// TIA Portal V17 export
// export: Created 2026-05-13T16:54:41.5069404Z, ExportSetting WithDefaults, DisplayName Totally Integrated Automation Portal, DisplayVersion V17 Update 4, DisplayName TIA Portal Openness, DisplayVersion V17 Update 4, DisplayName TIA Portal Version Control Interface, DisplayVersion V17, DisplayName SINAMICS Startdrive Advanced, DisplayVersion V17, DisplayName SINAMICS Startdrive G130, G150, S120, S150, SINAMICS MV, S210, DisplayVersion V17, DisplayName SINAMICS Startdrive G110M, G120, G120C, G120D, G120P, G115D, DisplayVersion V17, DisplayName STEP 7 Professional, DisplayVersion V17 Update 4, DisplayName STEP 7 Safety, DisplayVersion V17, DisplayName WinCC Professional, DisplayVersion V17 Update 4
TagTable "SV"
  SV_BD布袋压差高报 : Real  (PLC tag SV.BD布袋压差高报, HMI_连接_1, 1 s)
  SV_BD布袋压差高高报 : Real  (PLC tag SV.BD布袋压差高高报, HMI_连接_1, 1 s)
  SV_GX高效压差高报 : Real  (PLC tag SV.GX高效压差高报, HMI_连接_1, 1 s)
  SV_GX高效压差高高报 : Real  (PLC tag SV.GX高效压差高高报, HMI_连接_1, 1 s)
  SV_TN塔内压力高高报 : Real  (PLC tag SV.TN塔内压力高高报, HMI_连接_1, 1 s)
  SV_TN塔内压力低报 : Real  (PLC tag SV.TN塔内压力低报, HMI_连接_1, 1 s)
  SV_TN塔内压力低低报 : Real  (PLC tag SV.TN塔内压力低低报, HMI_连接_1, 1 s)
  SV_JL进料泵频率设定 : Real  (PLC tag SV.JL进料泵频率设定, HMI_连接_1, 1 s)
  SV_JF进风温度设定 : Real  (PLC tag SV.JF进风温度设定, HMI_连接_1, 1 s)
  SV_JF进温高报 : Real  (PLC tag SV.JF进温高报, HMI_连接_1, 1 s)
  SV_JF进温高高报 : Real  (PLC tag SV.JF进温高高报, HMI_连接_1, 1 s)
  SV_CF出风温度设定 : Real  (PLC tag SV.CF出风温度设定, HMI_连接_1, 1 s)
  SV_CF出温高报 : Real  (PLC tag SV.CF出温高报, HMI_连接_1, 1 s)
  SV_CF出温高高报 : Real  (PLC tag SV.CF出温高高报, HMI_连接_1, 1 s)
  SV_RS热水炉高报 : Real  (PLC tag SV.RS热水炉高报, HMI_连接_1, 1 s)
  SV_RS热水炉高高报 : Real  (PLC tag SV.RS热水炉高高报, HMI_连接_1, 1 s)
  SV_RS热水炉回收高报 : Real  (PLC tag SV.RS热水炉回收高报, HMI_连接_1, 1 s)
  SV_RS热水炉回收高高报 : Real  (PLC tag SV.RS热水炉回收高高报, HMI_连接_1, 1 s)
  SV_BD布袋反吹时间 : Real  (PLC tag SV.BD布袋反吹时间, HMI_连接_1, 1 s)
  SV_ZT主塔气锤时间 : Real  (PLC tag SV.ZT主塔气锤时间, HMI_连接_1, 1 s)
  SV_ZT主塔气扫时间 : Real  (PLC tag SV.ZT主塔气扫时间, HMI_连接_1, 1 s)
  SV_TN塔内压力高报 : Real  (PLC tag SV.TN塔内压力高报, HMI_连接_1, 1 s)
  SV_PM屏幕编号 : Real  (PLC tag SV.PM屏幕编号, HMI_连接_1, 1 s)
  SV_YQ氧气浓度 : Real  (PLC tag SV.YQ氧气浓度, HMI_连接_1, 1 s)
  SV_JF进风保护温度 : Real  (PLC tag SV.JF进风保护温度, HMI_连接_1, 1 s)
  SV_LX离心雾化 : Real  (PLC tag SV.LX离心雾化, HMI_连接_1, 1 s)
  SV_BD布袋振打时间 : Real  (PLC tag SV.BD布袋振打时间, HMI_连接_1, 1 s)
  SV_ZT主塔压力设定 : Real  (PLC tag SV.ZT主塔压力设定, HMI_连接_1, 1 s)
  SV_KQ空气流量设定 : Real  (PLC tag SV.KQ空气流量设定, HMI_连接_1, 1 s)
  SV_JL进料流量设定 : Real  (PLC tag SV.JL进料流量设定, HMI_连接_1, 1 s)
  SV_JF进风流量设定 : Real  (PLC tag SV.JF进风流量设定, HMI_连接_1, 1 s)
  SV_YF引风频率自动设定 : Real  (PLC tag SV.YF引风频率自动设定, HMI_连接_1, 1 s)
  SV_JL进料频率自动设定 : Real  (PLC tag SV.JL进料频率自动设定, HMI_连接_1, 1 s)
  SV_GX高效压差低报 : Real  (PLC tag SV.GX高效压差低报, HMI_连接_1, 1 s)
  SV_BD布袋压差低报 : Real  (PLC tag SV.BD布袋压差低报, HMI_连接_1, 1 s)
  SV_YF引风机频率设定 : Real  (PLC tag SV.YF引风机频率设定, HMI_连接_1, 1 s)
  SV_RS热水炉温度 : Real  (PLC tag SV.RS热水炉温度, HMI_连接_1, 1 s)
  SV_HW恒温系统温度 : Real  (PLC tag SV.HW恒温系统温度, HMI_连接_1, 1 s)
